FUNCTION_BLOCK FlushGritScreens (* CAT Function Block Type *)
  (* Standard: 61499-2 *)
  (* Version 0.0, 6/19/2026, Schneider Electric, template *)
  PACKAGE SE.Nereda;
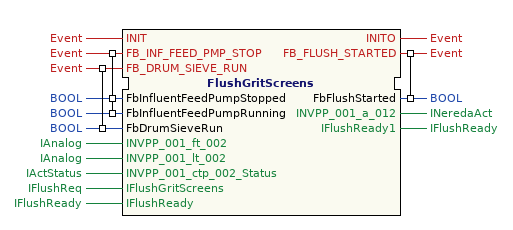
  EVENT_INPUT
    INIT;
    FB_INF_FEED_PMP_STOP WITH FbInfluentFeedPumpStopped, FbInfluentFeedPumpRunning;
    FB_DRUM_SIEVE_RUN WITH FbDrumSieveRun;
  END_EVENT
  EVENT_OUTPUT
    INITO;
    FB_FLUSH_STARTED WITH FbFlushStarted;
  END_EVENT
  VAR_INPUT
    FbInfluentFeedPumpStopped : BOOL;
    FbInfluentFeedPumpRunning : BOOL;
    FbDrumSieveRun : BOOL;
  END_VAR
  VAR_OUTPUT
    FbFlushStarted : BOOL;
  END_VAR
  SOCKETS
    INVPP_001_ft_002 : IAnalog;
    INVPP_001_lt_002 : IAnalog;
    INVPP_001_ctp_002_Status : IActStatus;
    IFlushGritScreens : IFlushReq;
    IFlushReady : IFlushReady;
  END_SOCKETS
  PLUGS
    INVPP_001_a_012 : INeredaAct;
    IFlushReady1 : IFlushReady;
  END_PLUGS
  (* 01 - FUNCTIONNAL INPUT INTERFACE *)
  (* 00 - INITIALIZATION *)
  (* 05 - LOGIC *)
  (* 06 - HMI INTERFACE *)
  (* 03 - FIELD INTERFACE *)
  (* Grit Screens Flush Conditions *)
  (* 02 - FUNCTIONNAL OUTPUT INTERFACE *)
  (* Grit Screens Flush Control *)
  FBS
    FlushConditions : FlushCdt(pin_AD4F1D04748929A2 := 'Effluent Level is ok', pin_D80C7C0ABBECCDAB := 'Grit Screen Installation Flushing', pin_2D24E9AB41BE5BDB := TRUE, pin_EDFD852BF7F500FC := '', pin_E55C299A5BCFE2A5 := 'NVPP 001 a-- 012 is Available', pin_4F5AA965534A9167 := 'No Low Low Flow Alarm (Effluent Pump)', pin_D8438E8592CCBB68 := 'Effluent Pump is Ready', pin_F9CA602A9987631B := 'Flushing Parametrization is Done', pin_D946781DFBE190E0 := 'Drum Sieve Motor Running', pin_2F47EB70426E0A5E := 'GS Installation Flushing Not Ready');
    IThis : FlushGritScreens_HMI(QI := TRUE);
    NVPP_001_lt_002_Status : decodeStatus; {SET_ATTRIBUTE(Configuration.Component.HideUnusedPorts, )}
    NotLowLevel : NOT_42C76073DCEB1A7A; {SET_ATTRIBUTE(Configuration.GenericFBType.InterfaceParams, Runtime.Standard#CNT:=1;OUT${CNT$}:BOOL)}
    GritScreensFlushControl : FlushingManagerGSs;
    CycleTime : E_DELAY_V_D;
    DurationTime : E_DELAY_V_D;
    Valve016_002Cmd : boolValueChanged;
    DurationSp : COMPARE_231D1C451B8C01CD0(IN2 := T#0ms); {SET_ATTRIBUTE(Configuration.GenericFBType.InterfaceParams, Runtime.Standard#CNT:=2;IN${CNT$}:TIME)} {SET_ATTRIBUTE(Configuration.Component.HideUnusedPorts, )}
    CycleSp : COMPARE_231D1C451B8C01CD0(IN2 := T#0ms); {SET_ATTRIBUTE(Configuration.GenericFBType.InterfaceParams, Runtime.Standard#CNT:=2;IN${CNT$}:TIME)} {SET_ATTRIBUTE(Configuration.Component.HideUnusedPorts, )}
    ConfigDone : AND_550FE6D62F509EB3; {SET_ATTRIBUTE(Configuration.GenericFBType.InterfaceParams, Runtime.Standard#CNT:=3;OUT:BOOL)}
    NVPP_001_ft_002_Status : decodeStatus; {SET_ATTRIBUTE(Configuration.Component.HideUnusedPorts, )}
    NotLowLowFlow : NOT_42C76073DCEB1A7A; {SET_ATTRIBUTE(Configuration.GenericFBType.InterfaceParams, Runtime.Standard#CNT:=1;OUT${CNT$}:BOOL)}
    CmdValve016_002 : BOOL2INT;
    FlowSp : COMPARE_1329C2AB45109BAAB(IN2 := 0); {SET_ATTRIBUTE(Configuration.GenericFBType.InterfaceParams, Runtime.Standard#CNT:=2;IN${CNT$}:REAL)} {SET_ATTRIBUTE(Configuration.Component.HideUnusedPorts, )}
    ForceStopSmooth : boolValueChanged;
    ForceStop : OR_NOT(pin_5391A9290C426EAD := FALSE, pin_0C6244A1FA53F771 := FALSE, pin_C718A4E0F6B1A5AF := FALSE, pin_F9B6B2F79CE46D8A := FALSE, pin_892061249439E371 := FALSE, pin_A17BF02B1ECA9592 := FALSE, pin_8BCAE36E149A36F2 := FALSE, pin_58FCE90E3A313BCD := TRUE, pin_7433DE8044744DCF := FALSE, pin_8555750E45CD1B5C := TRUE);
    ResetBtns : RESET_BTNs;
    GSInstNotReady : NOT_42C76073DCEB1A7A; {SET_ATTRIBUTE(Configuration.GenericFBType.InterfaceParams, Runtime.Standard#CNT:=1;OUT${CNT$}:BOOL)}
    Wait : E_DELAY(DT := T#2s);
  END_FBS
  EVENT_CONNECTIONS
    INVPP_001_lt_002.REQ_STATUS TO NVPP_001_lt_002_Status.REQ;
    NVPP_001_lt_002_Status.CNF TO NotLowLevel.REQ;
    FB_DRUM_SIEVE_RUN TO NotLowLevel.REQ;
    NotLowLowFlow.CNF TO DurationSp.REQ;
    DurationSp.CNF TO CycleSp.REQ;
    INVPP_001_ft_002.REQ_STATUS TO NVPP_001_ft_002_Status.REQ;
    NVPP_001_ft_002_Status.CNF TO NotLowLevel.REQ;
    NotLowLevel.CNF TO NotLowLowFlow.REQ;
    FlushConditions.E74FDFC5C9E17061 TO INITO;
    DurationTime.INITO TO FlushConditions.7689825C23C7E3C1;
    INVPP_001_a_012.9CD053F8408797ED TO GritScreensFlushControl.17EF565317C21577;
    CycleTime.1457E63E0C241C83 TO GritScreensFlushControl.FBAA1623341050FE;
    DurationTime.1457E63E0C241C83 TO GritScreensFlushControl.6BFDB43937C58B53;
    GritScreensFlushControl.FB17218C6899B6C2 TO FB_FLUSH_STARTED;
    GritScreensFlushControl.7C8478AB3E0AC40C TO Valve016_002Cmd.REQ;
    GritScreensFlushControl.4439D0346679ABD7 TO IFlushGritScreens.058C8BB5EF4C4954;
    GritScreensFlushControl.CNF_CYCLE_START TO CycleTime.START;
    GritScreensFlushControl.CNF_CYCLE_STOP TO CycleTime.STOP;
    GritScreensFlushControl.CNF_FLUSH_START TO DurationTime.START;
    GritScreensFlushControl.CNF_FLUSH_STOP TO DurationTime.STOP;
    Valve016_002Cmd.CHD TO CmdValve016_002.DD5870AA881150BB;
    CycleTime.INITO TO DurationTime.INIT;
    CmdValve016_002.6FC99A5BD1C38561 TO INVPP_001_a_012.0F1CDF9A9B4A227A;
    INVPP_001_a_012.CC753684FA882790 TO NotLowLevel.REQ;
    ForceStopSmooth.CNF TO FlushConditions.C4A26A2931936C6C;
    CycleSp.CNF TO FlowSp.REQ;
    FlowSp.CNF TO ConfigDone.REQ;
    ForceStop.5E2BC6C1897CC372 TO ForceStopSmooth.REQ;
    ConfigDone.CNF TO ForceStop.AE1B4DCC5DF54611;
    FB_INF_FEED_PMP_STOP TO GritScreensFlushControl.5E4003346E57F6E6;
    FlushConditions.144BD964598CDC30 TO GritScreensFlushControl.D472A6751679CB56;
    INIT TO IThis.1EF99DCB15A49BE4;
    GritScreensFlushControl.GRAPH TO IThis.623B20E659F013A2;
    FlushConditions.E74FDFC5C9E17061 TO IThis.6CA585F7EA2251CC;
    ResetBtns.920962203CA54948 TO IThis.BC4D95AF9C39047B;
    IThis.97A2502A32C860AE TO CycleTime.INIT;
    IThis.40B0BCBFC46CBB6D TO NotLowLevel.REQ;
    IThis.40B0BCBFC46CBB6D TO IFlushGritScreens.A591EFC748C65FB0;
    IThis.40B0BCBFC46CBB6D TO CycleTime.8C325F07198FCB13;
    IThis.40B0BCBFC46CBB6D TO DurationTime.8C325F07198FCB13;
    IThis.C0957A1C40CEA3B4 TO GritScreensFlushControl.F40A51463574875E;
    IThis.C0957A1C40CEA3B4 TO ResetBtns.AB695E9A35A20E19;
    GritScreensFlushControl.F622B0785D87399D TO IFlushGritScreens.91C62E5F9EC3AD97;
    INVPP_001_ctp_002_Status.14377629A1F197A9 TO NotLowLevel.REQ;
    IFlushGritScreens.158ACCEF11EA11F4 TO GritScreensFlushControl.2E9E428AF53DA484;
    IFlushReady.EB400628E9D6A506 TO GSInstNotReady.REQ;
    GSInstNotReady.CNF TO NotLowLevel.REQ;
    GritScreensFlushControl.F622B0785D87399D TO IFlushReady1.EB400628E9D6A506;
    FlushConditions.E74FDFC5C9E17061 TO IFlushReady1.EB400628E9D6A506;
    GritScreensFlushControl.ECD6779766443CCE TO Wait.START;
    Wait.EO TO GritScreensFlushControl.D6D3C004F4BF5676;
    INVPP_001_a_012.9CD053F8408797ED TO IFlushReady1.A6EF038FCF65FFCE;
    IFlushReady.A6EF038FCF65FFCE TO GritScreensFlushControl.E1B36525C625991C;
  END_CONNECTIONS
  DATA_CONNECTIONS
    INVPP_001_lt_002.Status TO NVPP_001_lt_002_Status.Status;
    NVPP_001_lt_002_Status.LoAlarm TO NotLowLevel.IN1;
    INVPP_001_ft_002.Status TO NVPP_001_ft_002_Status.Status;
    NVPP_001_ft_002_Status.LoLoAlarm TO NotLowLowFlow.IN1;
    NotLowLevel.OUT1 TO FlushConditions.22A84A30EE8DD605;
    INVPP_001_a_012.8A8A07EFCDA1443C TO FlushConditions.4ED40FD24D2392DA;
    NotLowLowFlow.OUT1 TO FlushConditions.504E64E2CDCF5D86;
    INVPP_001_ctp_002_Status.9E0B44559326BEAF TO FlushConditions.9BB2492C130556E4;
    FbDrumSieveRun TO FlushConditions.4E3CFAB7818DC81F;
    GritScreensFlushControl.7925856953128FBE TO FbFlushStarted;
    GritScreensFlushControl.6EFD4A5711C4475D TO Valve016_002Cmd.Input;
    GritScreensFlushControl.D35FF54DD8CD3DCD TO IFlushGritScreens.78ED129B4768A8A1;
    GritScreensFlushControl.809D6A4978DE08CF TO IFlushGritScreens.23612E77D592C190;
    Valve016_002Cmd.Output TO CmdValve016_002.4573FC8F228EB71D;
    CycleTime.716D3F3042596C89 TO GritScreensFlushControl.CycleTimeDone;
    DurationTime.716D3F3042596C89 TO GritScreensFlushControl.FlushDurationDone;
    INVPP_001_a_012.7F6CC7FEB9223DF3 TO GritScreensFlushControl.B4CCB3C919A81AAD;
    INVPP_001_a_012.A8D6C4A1FDCCA991 TO GritScreensFlushControl.927265D5AE017F25;
    IFlushGritScreens.309BBEDA7DF51DE0 TO GritScreensFlushControl.EB78D4EC51374885;
    IFlushGritScreens.E3447F193E0C5923 TO GritScreensFlushControl.8C9A5C84A4BBC11A;
    IFlushGritScreens.102FEFFE81A835E5 TO GritScreensFlushControl.BE830E3A77806910;
    IFlushGritScreens.32E78DF7D9CBD985 TO GritScreensFlushControl.CA6B1E62BFF3D73B;
    CmdValve016_002.A6DEF5F9C27C1848 TO INVPP_001_a_012.710D7FC54EE3F35A;
    DurationSp.NE TO ConfigDone.IN1;
    CycleSp.NE TO ConfigDone.IN2;
    ConfigDone.OUT TO FlushConditions.9D55FD7AD1246DA2;
    FlowSp.NE TO ConfigDone.IN3;
    ForceStop.39A6EB2EA34CB8B9 TO ForceStopSmooth.Input;
    NotLowLevel.OUT1 TO ForceStop.305F82B0106D312B;
    INVPP_001_a_012.8A8A07EFCDA1443C TO ForceStop.DD1680AE8DA8DF87;
    NotLowLowFlow.OUT1 TO ForceStop.92ECDEDDB24CC262;
    INVPP_001_ctp_002_Status.9E0B44559326BEAF TO ForceStop.2CF1E7F52666F162;
    ConfigDone.OUT TO ForceStop.4997B302A4472F6A;
    FbInfluentFeedPumpStopped TO GritScreensFlushControl.A7C5B43F7896B8B7;
    FbInfluentFeedPumpRunning TO GritScreensFlushControl.AC6BF7D02159B6C4;
    FlushConditions.5C1922DA22925005 TO GritScreensFlushControl.EnableOperation;
    GritScreensFlushControl.Grafcet TO IThis.4EF02231C06E8D13;
    IThis.16EEFB003671CC3A TO CycleSp.IN1;
    IThis.16EEFB003671CC3A TO CycleTime.DT1;
    IThis.1AA6078AD289AF22 TO DurationSp.IN1;
    IThis.1AA6078AD289AF22 TO DurationTime.DT1;
    IThis.3E1384426DD858B0 TO FlowSp.IN1;
    IThis.3E1384426DD858B0 TO IFlushGritScreens.34B76CCA964D89EE;
    IThis.CEC3C53B3ACE8E6D TO GritScreensFlushControl.0FA765E9822F7BA9;
    IThis.CEC3C53B3ACE8E6D TO ResetBtns.479D4538AEFD6EE1;
    IThis.1BFB680DD0A7C843 TO GritScreensFlushControl.3C22F17908DBA162;
    GritScreensFlushControl.51D0A2C29DC62FA2 TO IFlushGritScreens.B5CD30493D22784A;
    GritScreensFlushControl.7AB11AE4573B259E TO IFlushGritScreens.10050E1891596878;
    IFlushGritScreens.0154EF4D281C90FC TO GritScreensFlushControl.9CD632B5AC2CF415;
    IFlushReady.948E4422D799D3D4 TO GSInstNotReady.IN1;
    GSInstNotReady.OUT1 TO FlushConditions.47969CBC2D520AAD;
    GritScreensFlushControl.51D0A2C29DC62FA2 TO IFlushReady1.948E4422D799D3D4;
    IFlushGritScreens.F75B2D6279DB7772 TO GritScreensFlushControl.5E80D184B53E9B75;
    IFlushGritScreens.FBD19C5680BE3A13 TO GritScreensFlushControl.F178DB7E20F3649C;
    INVPP_001_a_012.7F6CC7FEB9223DF3 TO IFlushReady1.3B406C848FF944CA;
    IFlushReady.3B406C848FF944CA TO GritScreensFlushControl.248BD6B0D63F5917;
  END_CONNECTIONS
END_FUNCTION_BLOCK
